Fanuc KAREL source: compact_preamble.KL

PROGRAM KT00958
%NOLOCKGROUP
VAR
ENTRY:INTEGER;PNAME : STRING[80];VNAME : STRING[80];STATUS:INTEGER;VALUE:BOOLEAN
BEGIN
ENTRY=0
PNAME=''
VNAME='VALUE'
SET_VAR(ENTRY,PNAME,VNAME,VALUE,STATUS)
END KT00958
